(* Logix 5000 project; controller Y059_LHM vendor 1 type 14 code 156 rev 32.13; software revision 32.00 *)

TASK MainTask (periodic, rate 100 ms, priority 5, watchdog 500 ms) : MainProgram

MODULES
   Local : vendor 1 type 14 code 156 (Compact 0, rev 32.13)
      Module1 : 1769-IQ16 (Compact 1, rev 1.1, Input RPI 20 ms)
      Module2 : 1769-OB16 (Compact 2, rev 2.1, Output RPI 20 ms)
      SIC_101_Kinetix : vendor 1 type 37 code 50 (Ethernet 10.1.5.59, rev 7.11, MotionSync RPI 2 ms, MotionDiagnostics RPI 1 ms)
      SIC_201_Kinetix : vendor 1 type 37 code 50 (Ethernet 10.1.5.60, rev 7.1, MotionSync RPI 2 ms, MotionDiagnostics RPI 1 ms)
      Stratix5700 : vendor 1 type 12 code 242 (Ethernet 10.1.5.253, rev 10.1, Output RPI 1000 ms)
END_MODULES

TYPE Command :
STRUCT
   Command : DINT;   // 0=Run, 1=Fault Reset,
   Speed : REAL;   // Speed
END_STRUCT
END_TYPE

TYPE CommInfo :
STRUCT
   BoolTags : DINT;
   HeartBeat : DINT;
END_STRUCT
END_TYPE

TYPE FaultRecord :
STRUCT
   TimeLow : DINT;
   TimeHigh : DINT;
   Type : INT;
   Code : INT;
   Info : DINT[8];
END_STRUCT
END_TYPE

TYPE PumpController :
STRUCT
   RunCMD : BOOL;   // Run Command
   ResetCMD : BOOL;   // Reset Command
   isFaulted : BOOL;   // Fault Status, (0= Not Fault, 1= Faulted)
   isRunning : BOOL;   // Run Status, (0=Stopped, 1=Running)
   isServoOK : BOOL;   // Communications between the PLC and Servo (0=Not OK, 1=OK)
   isPressureHigh : BOOL;   // Outlet Pressure High Status (0=Not High, 1=High)
   isDecontactor : BOOL;   // Decontactor from STO circuit( 0=Contact OK, 1= Not Contact)
   FautCode : DINT;   // Fault Code
   SpeedSP : SetPoint;   // Speed Setpoint
   SpeedFeedback : SetPoint;   // Speed Feedback
   Ok2Run : BOOL;   // OK to Run Pump
   ResetTimer : TIMER;   // Heart Beat Error Reset Timer
END_STRUCT
END_TYPE

TYPE SetPoint :
STRUCT
   Min : REAL;
   SP : REAL;
   Max : REAL;
END_STRUCT
END_TYPE

TYPE Status :
STRUCT
   Status : DINT;   // 0=isDecontacted, 1=isFaulted, 2=isPressureHigh, 3=isRunning, 4=isServoOK
   FaultCode : DINT;
   SpeedFdbk : REAL;
END_STRUCT
END_TYPE

ADD_ON_INSTRUCTION SERVO_AOI   (* revision 1.0, vendor Lewa Process Technologies *)
// Servo AOI
// Help:
// Version 1.0
// 18 May, 2018
VAR_IN_OUT
   CONTROLLER : PumpController; {required}
   DRIVE_AXIS : AXIS_CIP_DRIVE; {required}
END_VAR
VAR_INPUT
   GearBox_Ratio : REAL; {access Read Only, required}   // GearBox Ratio (Read from Pump Name Plate)
   Axis_AccDec : REAL := 20.0; {required}
   Pump_RPM_Max : DINT; {access Read Only, required}
   Pump_RPM_Min : DINT; {access None, required}
END_VAR
VAR_OUTPUT
   Pump_RPM_Val : REAL; {access Read Only, visible}
   Motor_RPS : REAL; {visible}   // Speed RPS
END_VAR
VAR
   Local_Axis_MAFR : MOTION_INSTRUCTION;
   Local_Axis_MAJ : MOTION_INSTRUCTION;
   Local_Axis_MAS : MOTION_INSTRUCTION;
   Local_Axis_MCD : MOTION_INSTRUCTION;
   Local_Axis_MSF : MOTION_INSTRUCTION;
   Local_Axis_MSO : MOTION_INSTRUCTION;
   Motor_RPS_Prev : REAL;   // Previous Speed RPS
   Local_Axis_Start : BOOL;   // Servo Start/Stop Command
   Local_1000MaxRPM : DINT;   // 1000 Times Max RPM
   Local_RunDelay : TIMER := (PRE := 2000);
   Local_1000RPM : DINT; {access None}   // 1000 Times RPM
   Local_1000MinRPM : DINT; {access None}   // 1000 Times Min RPM
   ServoActualRPS : REAL; {access None}
   ServoActual : DINT; {access None}   // Motor RPS for Feedback
   Feedbk_1000RPM : DINT; {access None}   // 1000 Times RPM for Feedback
   Axis_Last_TrackingNotchFilter : REAL; {access None}
   Axis_NotchFilter_Seq : DINT; {access None}
   Axis_Timer : TIMER[4] := ([0].PRE := 50, [0].ACC := 60, [1].PRE := 50); {access None}
   Axis_CountUP : DINT; {access None}
   Axis_ONS0 : BOOL; {access None}
   Axis_AdaptiveTuning_Mode : DINT; {access None}
   Motor_RPS_ONS : BOOL; {access None}
END_VAR

ROUTINE Logic   (* ladder *)
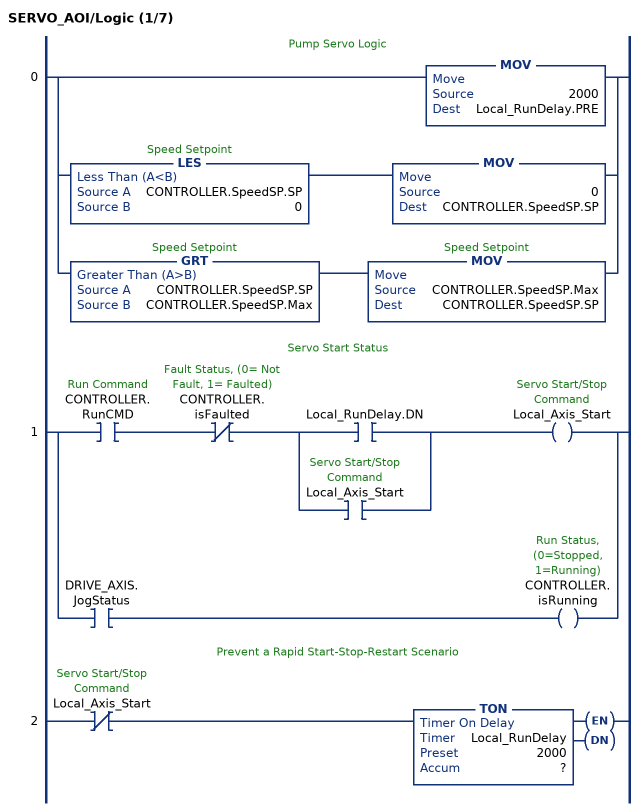
   // Pump Servo Logic
   0: [MOV(2000,Local_RunDelay.PRE) ,LES(CONTROLLER.SpeedSP.SP,0) MOV(0,CONTROLLER.SpeedSP.SP) ,GRT(CONTROLLER.SpeedSP.SP,CONTROLLER.SpeedSP.Max) MOV(CONTROLLER.SpeedSP.Max,CONTROLLER.SpeedSP.SP) ];
   // Servo Start Status
   1: [XIC(CONTROLLER.RunCMD) XIO(CONTROLLER.isFaulted) [XIC(Local_RunDelay.DN) ,XIC(Local_Axis_Start) ] OTE(Local_Axis_Start) ,XIC(DRIVE_AXIS.JogStatus) OTE(CONTROLLER.isRunning) ];
   // Prevent a Rapid Start-Stop-Restart Scenario
   2: XIO(Local_Axis_Start)TON(Local_RunDelay,?,?);
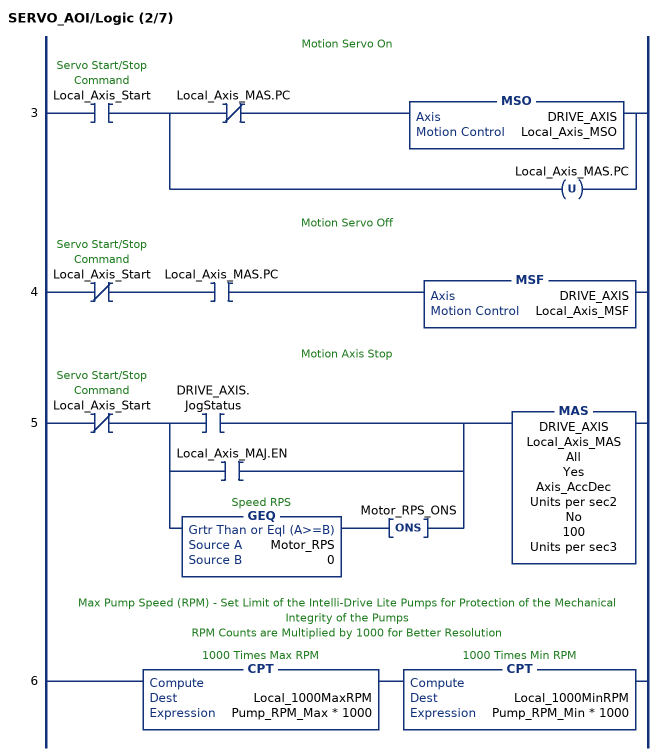
   // Motion Servo On
   3: XIC(Local_Axis_Start)[XIO(Local_Axis_MAS.PC) MSO(DRIVE_AXIS,Local_Axis_MSO) ,OTU(Local_Axis_MAS.PC) ];
   // Motion Servo Off
   4: XIO(Local_Axis_Start)XIC(Local_Axis_MAS.PC)MSF(DRIVE_AXIS,Local_Axis_MSF);
   // Motion Axis Stop
   5: XIO(Local_Axis_Start)[[XIC(DRIVE_AXIS.JogStatus) ,XIC(Local_Axis_MAJ.EN) ] ,GEQ(Motor_RPS,0) ONS(Motor_RPS_ONS) ]MAS(DRIVE_AXIS,Local_Axis_MAS,All,Yes,Axis_AccDec,Units per sec2,No,100,Units per sec3);
   // Max Pump Speed (RPM) - Set Limit of the Intelli-Drive Lite Pumps for Protection of the Mechanical Integrity of the Pumps
   // RPM Counts are Multiplied by 1000 for Better Resolution
   6: CPT(Local_1000MaxRPM,Pump_RPM_Max * 1000)CPT(Local_1000MinRPM,Pump_RPM_Min * 1000);
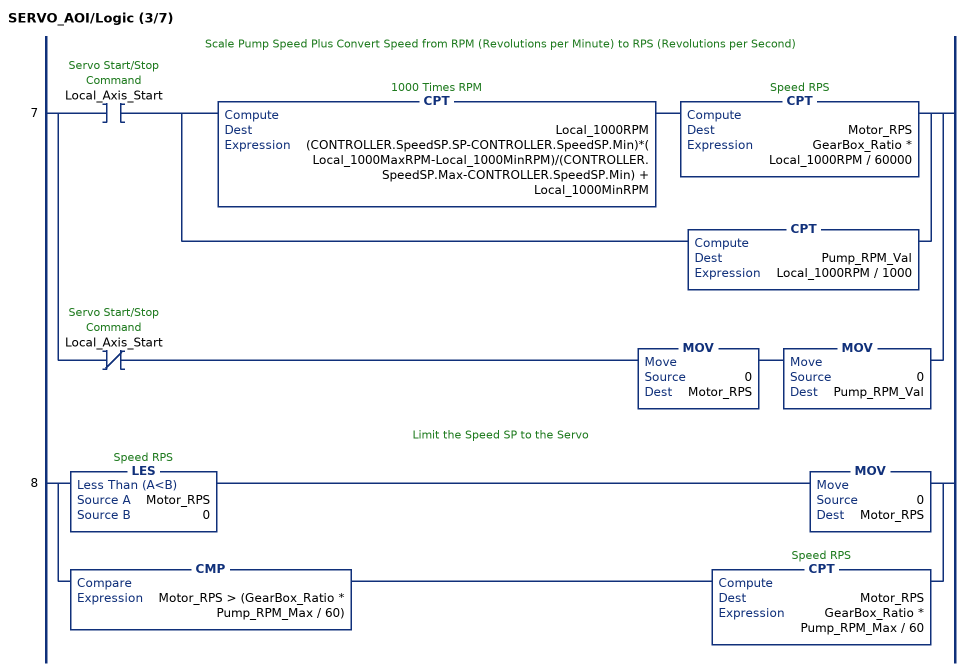
   // Scale Pump Speed Plus Convert Speed from RPM (Revolutions per Minute) to RPS (Revolutions per Second)
   7: [XIC(Local_Axis_Start) [CPT(Local_1000RPM,(CONTROLLER.SpeedSP.SP-CONTROLLER.SpeedSP.Min)*(Local_1000MaxRPM-Local_1000MinRPM)/(CONTROLLER.SpeedSP.Max-CONTROLLER.SpeedSP.Min) + Local_1000MinRPM) CPT(Motor_RPS,GearBox_Ratio * Local_1000RPM / 60000) ,CPT(Pump_RPM_Val,Local_1000RPM / 1000) ] ,XIO(Local_Axis_Start) MOV(0,Motor_RPS) MOV(0,Pump_RPM_Val) ];
   // Limit the Speed SP to the Servo
   8: [LES(Motor_RPS,0) MOV(0,Motor_RPS) ,CMP(Motor_RPS > (GearBox_Ratio * Pump_RPM_Max / 60)) CPT(Motor_RPS,GearBox_Ratio * Pump_RPM_Max / 60) ];
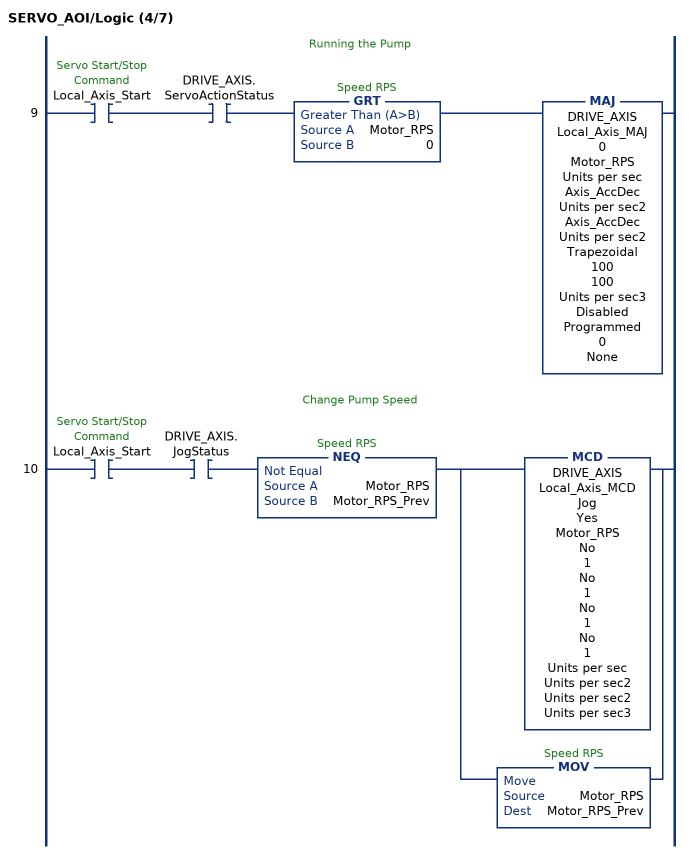
   // Running the Pump
   9: XIC(Local_Axis_Start)XIC(DRIVE_AXIS.ServoActionStatus)GRT(Motor_RPS,0)MAJ(DRIVE_AXIS,Local_Axis_MAJ,0,Motor_RPS,Units per sec,Axis_AccDec,Units per sec2,Axis_AccDec,Units per sec2,Trapezoidal,100,100,Units per sec3,Disabled,Programmed,0,None);
   // Change Pump Speed
   10: XIC(Local_Axis_Start)XIC(DRIVE_AXIS.JogStatus)NEQ(Motor_RPS,Motor_RPS_Prev)[MCD(DRIVE_AXIS,Local_Axis_MCD,Jog,Yes,Motor_RPS,No,1,No,1,No,1,No,1,Units per sec,Units per sec2,Units per sec2,Units per sec3) ,MOV(Motor_RPS,Motor_RPS_Prev) ];
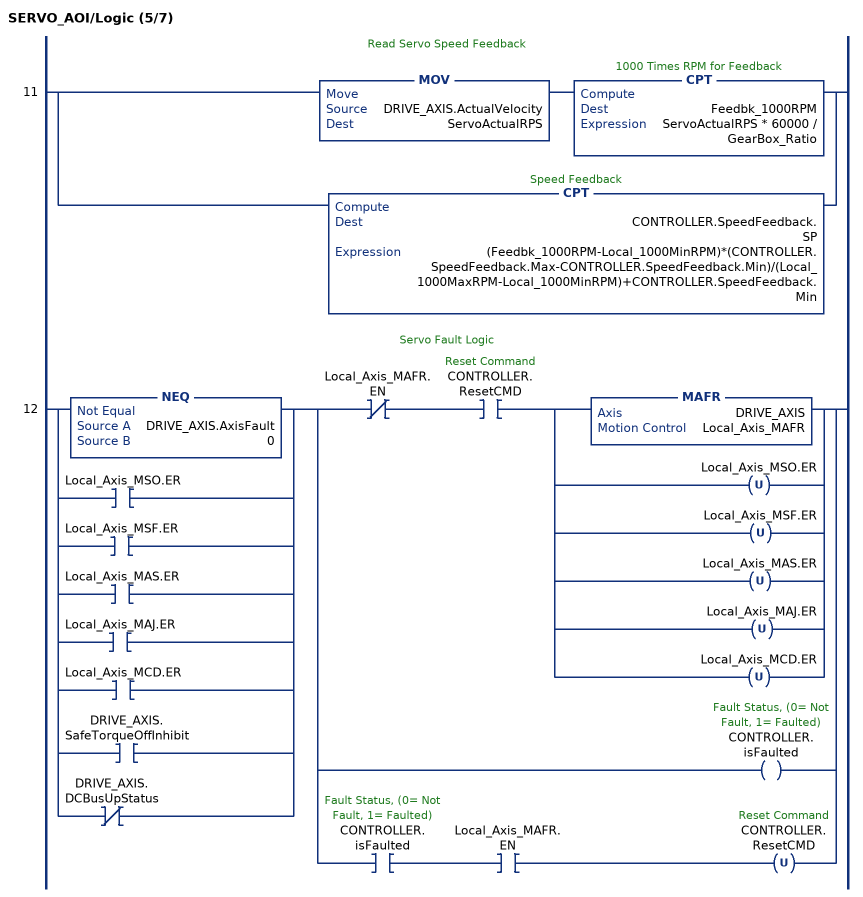
   // Read Servo Speed Feedback
   11: [MOV(DRIVE_AXIS.ActualVelocity,ServoActualRPS) CPT(Feedbk_1000RPM,ServoActualRPS * 60000 / GearBox_Ratio) ,CPT(CONTROLLER.SpeedFeedback.SP,(Feedbk_1000RPM-Local_1000MinRPM)*(CONTROLLER.SpeedFeedback.Max-CONTROLLER.SpeedFeedback.Min)/(Local_1000MaxRPM-Local_1000MinRPM)+CONTROLLER.SpeedFeedback.Min) ];
   // Servo Fault Logic
   12: [NEQ(DRIVE_AXIS.AxisFault,0) ,XIC(Local_Axis_MSO.ER) ,XIC(Local_Axis_MSF.ER) ,XIC(Local_Axis_MAS.ER) ,XIC(Local_Axis_MAJ.ER) ,XIC(Local_Axis_MCD.ER) ,XIC(DRIVE_AXIS.SafeTorqueOffInhibit) ,XIO(DRIVE_AXIS.DCBusUpStatus) ][XIO(Local_Axis_MAFR.EN) XIC(CONTROLLER.ResetCMD) [MAFR(DRIVE_AXIS,Local_Axis_MAFR) ,OTU(Local_Axis_MSO.ER) ,OTU(Local_Axis_MSF.ER) ,OTU(Local_Axis_MAS.ER) ,OTU(Local_Axis_MAJ.ER) ,OTU(Local_Axis_MCD.ER) ] ,OTE(CONTROLLER.isFaulted) ,XIC(CONTROLLER.isFaulted) XIC(Local_Axis_MAFR.EN) OTU(CONTROLLER.ResetCMD) ];
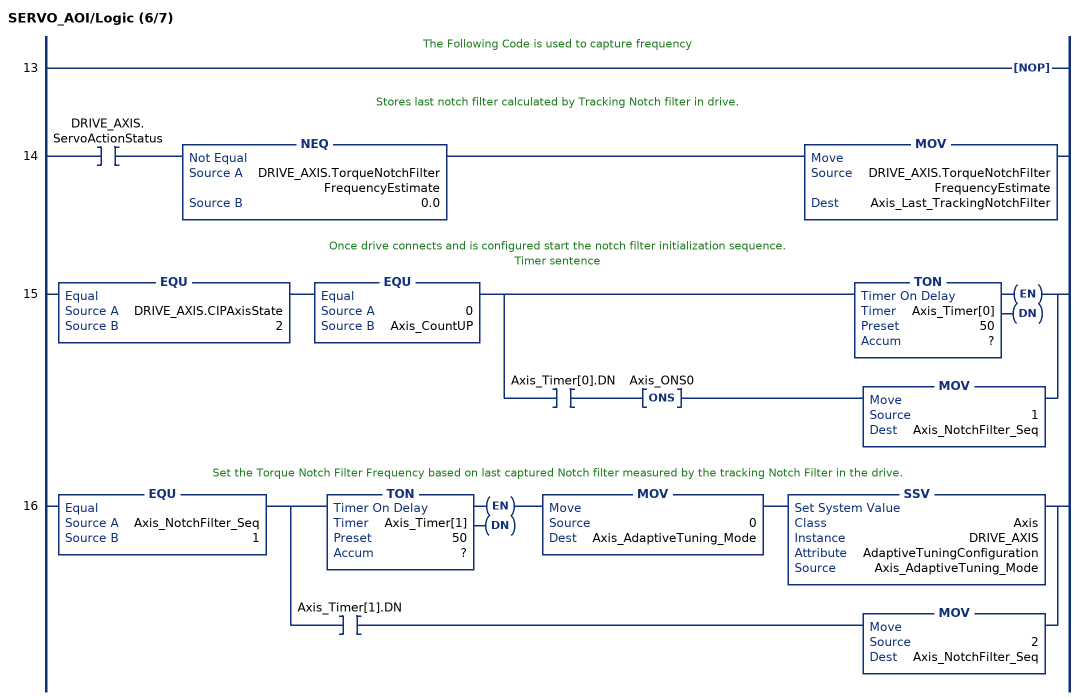
   // The Following Code is used to capture frequency
   13: NOP();
   // Stores last notch filter calculated by Tracking Notch filter in drive.
   14: XIC(DRIVE_AXIS.ServoActionStatus)NEQ(DRIVE_AXIS.TorqueNotchFilterFrequencyEstimate,0.0)MOV(DRIVE_AXIS.TorqueNotchFilterFrequencyEstimate,Axis_Last_TrackingNotchFilter);
   // Once drive connects and is configured start the notch filter initialization sequence.
   // Timer sentence
   15: EQU(DRIVE_AXIS.CIPAxisState,2)EQU(0,Axis_CountUP)[TON(Axis_Timer[0],?,?) ,XIC(Axis_Timer[0].DN) ONS(Axis_ONS0) MOV(1,Axis_NotchFilter_Seq) ];
   // Set the Torque Notch Filter Frequency based on last captured Notch filter measured by the tracking Notch Filter in the drive.
   16: EQU(Axis_NotchFilter_Seq,1)[TON(Axis_Timer[1],?,?) MOV(0,Axis_AdaptiveTuning_Mode) SSV(Axis,DRIVE_AXIS,AdaptiveTuningConfiguration,Axis_AdaptiveTuning_Mode) ,XIC(Axis_Timer[1].DN) MOV(2,Axis_NotchFilter_Seq) ];
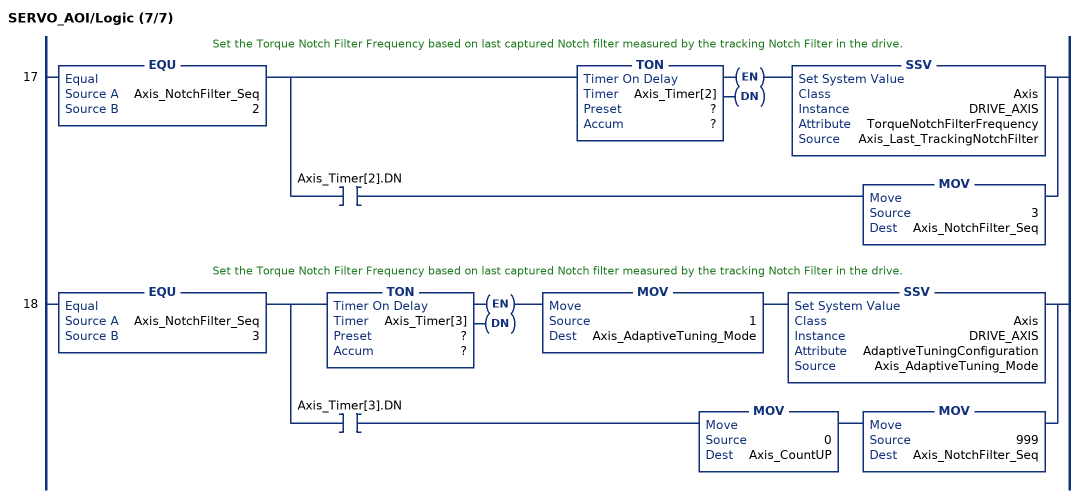
   // Set the Torque Notch Filter Frequency based on last captured Notch filter measured by the tracking Notch Filter in the drive.
   17: EQU(Axis_NotchFilter_Seq,2)[TON(Axis_Timer[2],?,?) SSV(Axis,DRIVE_AXIS,TorqueNotchFilterFrequency,Axis_Last_TrackingNotchFilter) ,XIC(Axis_Timer[2].DN) MOV(3,Axis_NotchFilter_Seq) ];
   // Set the Torque Notch Filter Frequency based on last captured Notch filter measured by the tracking Notch Filter in the drive.
   18: EQU(Axis_NotchFilter_Seq,3)[TON(Axis_Timer[3],?,?) MOV(1,Axis_AdaptiveTuning_Mode) SSV(Axis,DRIVE_AXIS,AdaptiveTuningConfiguration,Axis_AdaptiveTuning_Mode) ,XIC(Axis_Timer[3].DN) MOV(0,Axis_CountUP) MOV(999,Axis_NotchFilter_Seq) ];
END_ROUTINE
END_ADD_ON_INSTRUCTION

ADD_ON_INSTRUCTION ServoFaultCode   (* revision 1.0, vendor YMC Process Technologies *)
VAR_IN_OUT
   Axis_1 : AXIS_CIP_DRIVE; {required}
END_VAR
VAR_INPUT
   DriveConnStatus : DINT := 16#0000_4000; {required}
END_VAR
VAR_OUTPUT
   FaultCode : DINT; {access Read Only, required}
   FaultType : DINT; {access Read Only, required}
   LocalFaultDetected : BOOL; {access None, required}
END_VAR
VAR
   A1_CIPAxisFaultsLSW : DINT;
   A1_CIPAxisFaultsMSW : DINT := 45;
   A1_CIPAxisFaultsRA_LSW : DINT;
   A1_CIPAxisFaultsRA_MSW : DINT;
   ErrorCode : DINT[20] := ([1] := 8192);
   IntegratedSTOSxx : DINT; {access None}
   A1_AxisSafetyFaults : DINT; {access None}
   Drive_CommConnectionOK : BOOL; {access None}
   TempCipAxisFaultsRA : DINT[2]; {access None}
   ClearFault : DINT; {access None}
END_VAR

ROUTINE Logic   (* ladder *)
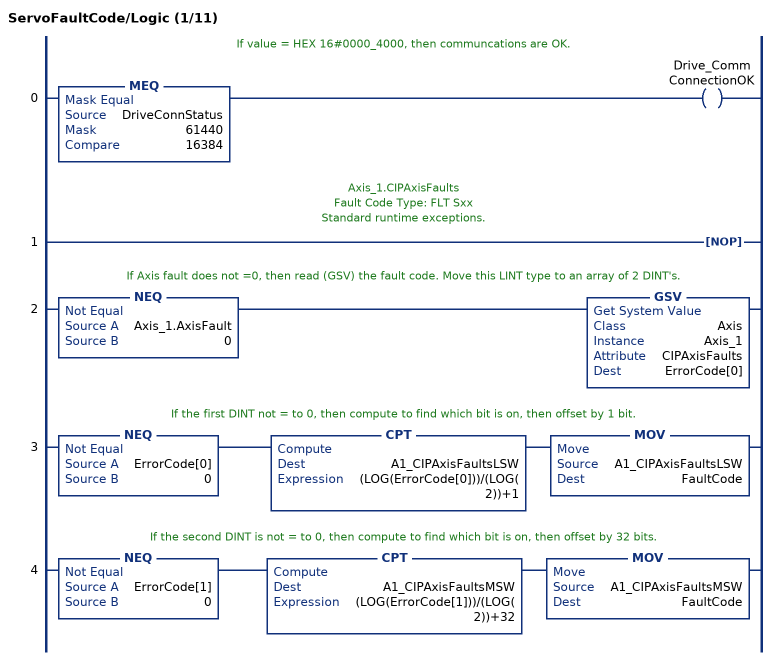
   // If value = HEX 16#0000_4000, then communcations are OK.
   0: MEQ(DriveConnStatus,61440,16384)OTE(Drive_CommConnectionOK);
   // Axis_1.CIPAxisFaults
   // Fault Code Type: FLT Sxx
   // Standard runtime exceptions.
   1: NOP();
   // If Axis fault does not =0, then read (GSV) the fault code. Move this LINT type to an array of 2 DINT's.
   2: NEQ(Axis_1.AxisFault,0)GSV(Axis,Axis_1,CIPAxisFaults,ErrorCode[0]);
   // If the first DINT not = to 0, then compute to find which bit is on, then offset by 1 bit.
   3: NEQ(ErrorCode[0],0)CPT(A1_CIPAxisFaultsLSW,(LOG(ErrorCode[0]))/(LOG(2))+1)MOV(A1_CIPAxisFaultsLSW,FaultCode);
   // If the second DINT is not = to 0, then compute to find which bit is on, then offset by 32 bits.
   4: NEQ(ErrorCode[1],0)CPT(A1_CIPAxisFaultsMSW,(LOG(ErrorCode[1]))/(LOG(2))+32)MOV(A1_CIPAxisFaultsMSW,FaultCode);
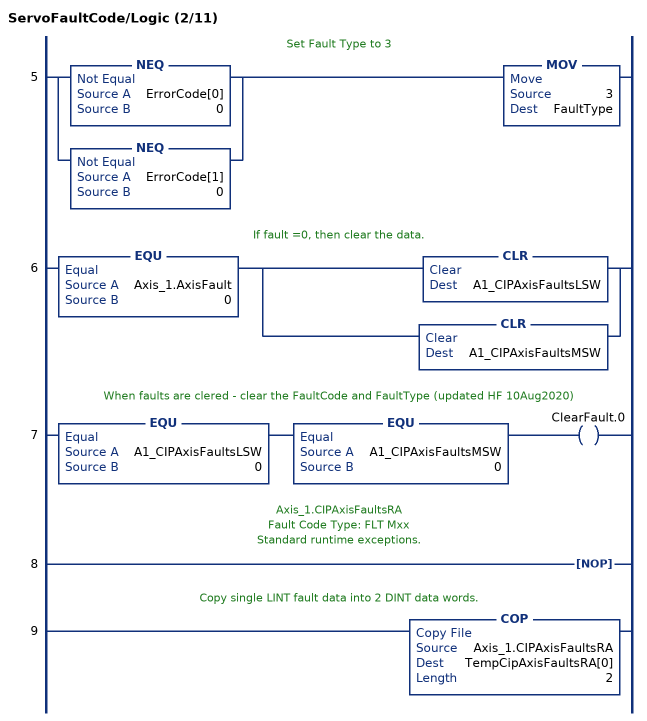
   // Set Fault Type to 3
   5: [NEQ(ErrorCode[0],0) ,NEQ(ErrorCode[1],0) ]MOV(3,FaultType);
   // If fault =0, then clear the data.
   6: EQU(Axis_1.AxisFault,0)[CLR(A1_CIPAxisFaultsLSW) ,CLR(A1_CIPAxisFaultsMSW) ];
   // When faults are clered - clear the FaultCode and FaultType (updated HF 10Aug2020)
   7: EQU(A1_CIPAxisFaultsLSW,0)EQU(A1_CIPAxisFaultsMSW,0)OTE(ClearFault.0);
   // Axis_1.CIPAxisFaultsRA
   // Fault Code Type: FLT Mxx
   // Standard runtime exceptions.
   8: NOP();
   // Copy single LINT fault data into 2 DINT data words.
   9: COP(Axis_1.CIPAxisFaultsRA,TempCipAxisFaultsRA[0],2);
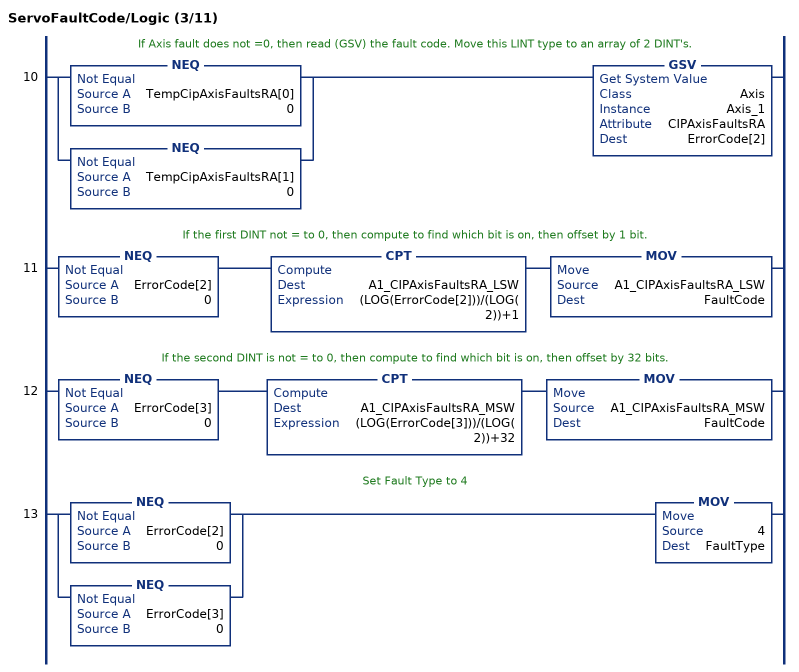
   // If Axis fault does not =0, then read (GSV) the fault code. Move this LINT type to an array of 2 DINT's.
   10: [NEQ(TempCipAxisFaultsRA[0],0) ,NEQ(TempCipAxisFaultsRA[1],0) ]GSV(Axis,Axis_1,CIPAxisFaultsRA,ErrorCode[2]);
   // If the first DINT not = to 0, then compute to find which bit is on, then offset by 1 bit.
   11: NEQ(ErrorCode[2],0)CPT(A1_CIPAxisFaultsRA_LSW,(LOG(ErrorCode[2]))/(LOG(2))+1)MOV(A1_CIPAxisFaultsRA_LSW,FaultCode);
   // If the second DINT is not = to 0, then compute to find which bit is on, then offset by 32 bits.
   12: NEQ(ErrorCode[3],0)CPT(A1_CIPAxisFaultsRA_MSW,(LOG(ErrorCode[3]))/(LOG(2))+32)MOV(A1_CIPAxisFaultsRA_MSW,FaultCode);
   // Set Fault Type to 4
   13: [NEQ(ErrorCode[2],0) ,NEQ(ErrorCode[3],0) ]MOV(4,FaultType);
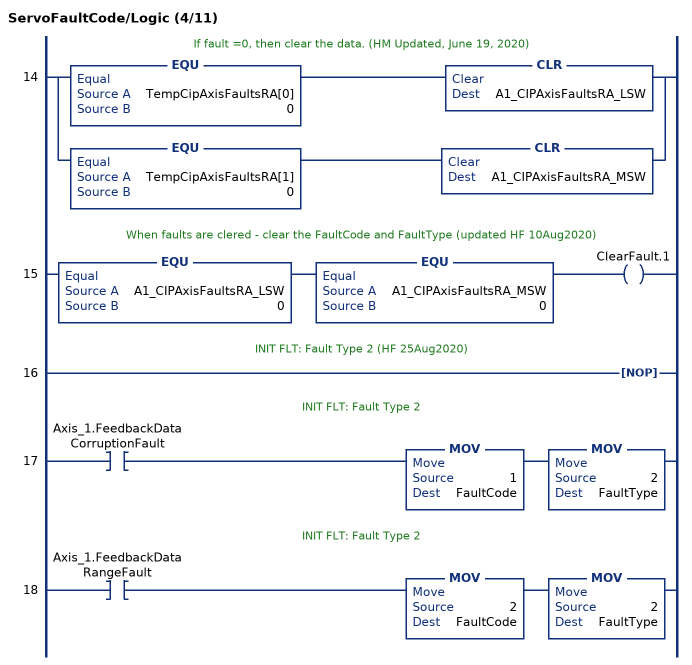
   // If fault =0, then clear the data. (HM Updated, June 19, 2020)
   14: [EQU(TempCipAxisFaultsRA[0],0) CLR(A1_CIPAxisFaultsRA_LSW) ,EQU(TempCipAxisFaultsRA[1],0) CLR(A1_CIPAxisFaultsRA_MSW) ];
   // When faults are clered - clear the FaultCode and FaultType (updated HF 10Aug2020)
   15: EQU(A1_CIPAxisFaultsRA_LSW,0)EQU(A1_CIPAxisFaultsRA_MSW,0)OTE(ClearFault.1);
   // INIT FLT: Fault Type 2 (HF 25Aug2020)
   16: NOP();
   // INIT FLT: Fault Type 2
   17: XIC(Axis_1.FeedbackDataCorruptionFault)MOV(1,FaultCode)MOV(2,FaultType);
   // INIT FLT: Fault Type 2
   18: XIC(Axis_1.FeedbackDataRangeFault)MOV(2,FaultCode)MOV(2,FaultType);
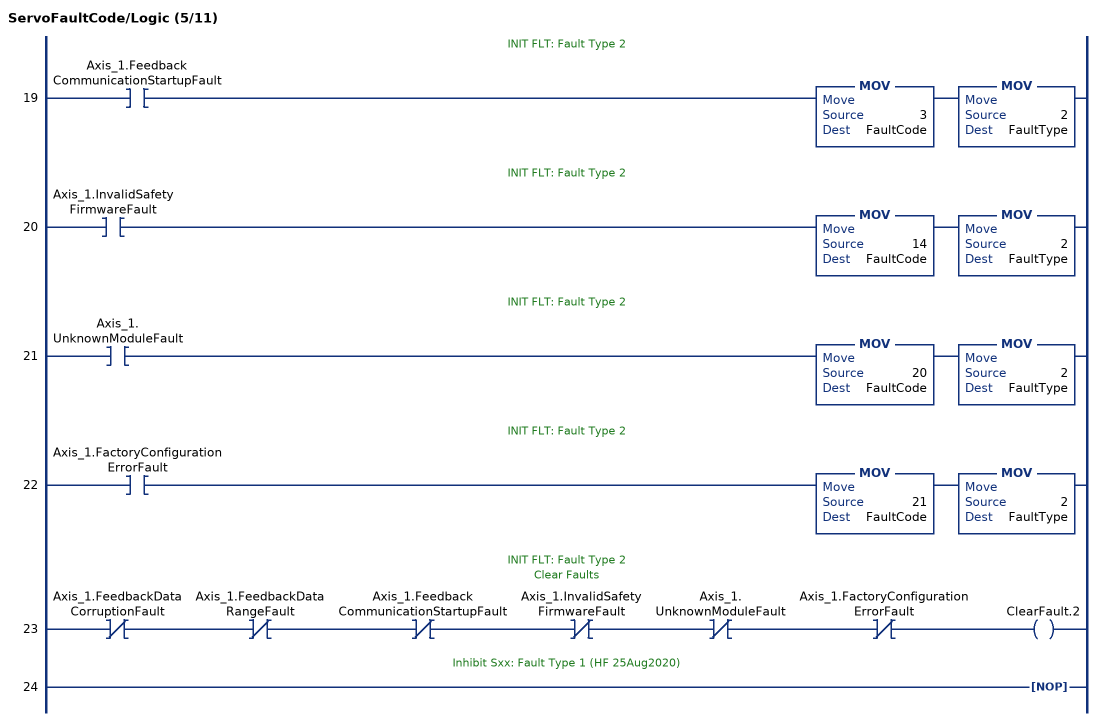
   // INIT FLT: Fault Type 2
   19: XIC(Axis_1.FeedbackCommunicationStartupFault)MOV(3,FaultCode)MOV(2,FaultType);
   // INIT FLT: Fault Type 2
   20: XIC(Axis_1.InvalidSafetyFirmwareFault)MOV(14,FaultCode)MOV(2,FaultType);
   // INIT FLT: Fault Type 2
   21: XIC(Axis_1.UnknownModuleFault)MOV(20,FaultCode)MOV(2,FaultType);
   // INIT FLT: Fault Type 2
   22: XIC(Axis_1.FactoryConfigurationErrorFault)MOV(21,FaultCode)MOV(2,FaultType);
   // INIT FLT: Fault Type 2
   // Clear Faults
   23: XIO(Axis_1.FeedbackDataCorruptionFault)XIO(Axis_1.FeedbackDataRangeFault)XIO(Axis_1.FeedbackCommunicationStartupFault)XIO(Axis_1.InvalidSafetyFirmwareFault)XIO(Axis_1.UnknownModuleFault)XIO(Axis_1.FactoryConfigurationErrorFault)OTE(ClearFault.2);
   // Inhibit Sxx: Fault Type 1 (HF 25Aug2020)
   24: NOP();
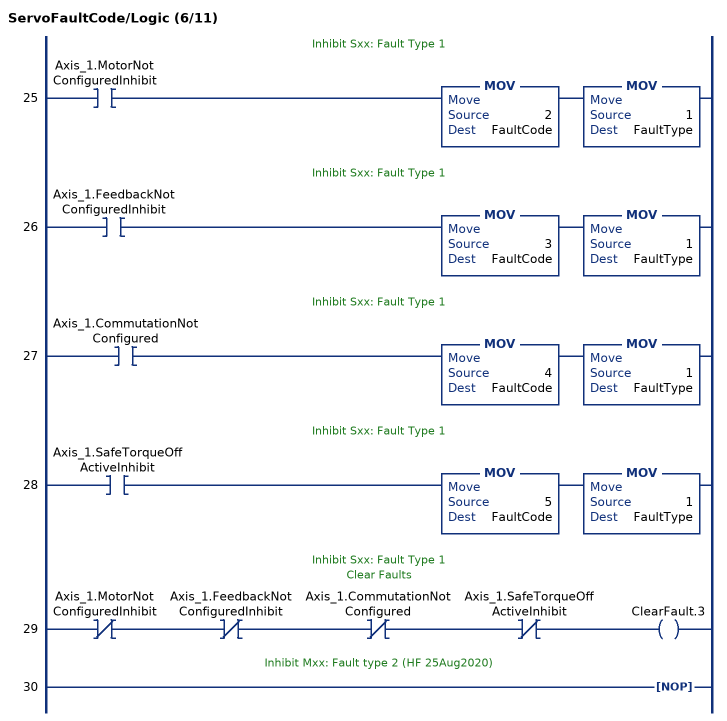
   // Inhibit Sxx: Fault Type 1
   25: XIC(Axis_1.MotorNotConfiguredInhibit)MOV(2,FaultCode)MOV(1,FaultType);
   // Inhibit Sxx: Fault Type 1
   26: XIC(Axis_1.FeedbackNotConfiguredInhibit)MOV(3,FaultCode)MOV(1,FaultType);
   // Inhibit Sxx: Fault Type 1
   27: XIC(Axis_1.CommutationNotConfigured)MOV(4,FaultCode)MOV(1,FaultType);
   // Inhibit Sxx: Fault Type 1
   28: XIC(Axis_1.SafeTorqueOffActiveInhibit)MOV(5,FaultCode)MOV(1,FaultType);
   // Inhibit Sxx: Fault Type 1
   // Clear Faults
   29: XIO(Axis_1.MotorNotConfiguredInhibit)XIO(Axis_1.FeedbackNotConfiguredInhibit)XIO(Axis_1.CommutationNotConfigured)XIO(Axis_1.SafeTorqueOffActiveInhibit)OTE(ClearFault.3);
   // Inhibit Mxx: Fault type 2 (HF 25Aug2020)
   30: NOP();
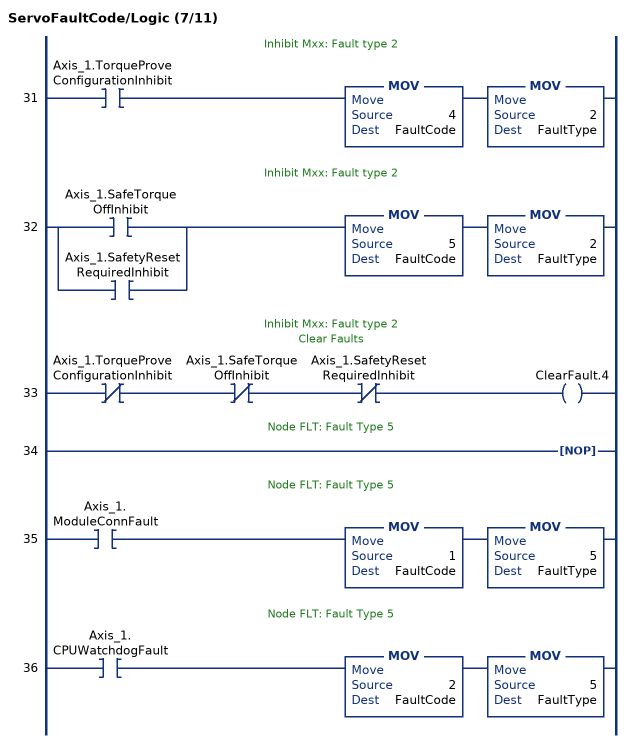
   // Inhibit Mxx: Fault type 2
   31: XIC(Axis_1.TorqueProveConfigurationInhibit)MOV(4,FaultCode)MOV(2,FaultType);
   // Inhibit Mxx: Fault type 2
   32: [XIC(Axis_1.SafeTorqueOffInhibit) ,XIC(Axis_1.SafetyResetRequiredInhibit) ]MOV(5,FaultCode)MOV(2,FaultType);
   // Inhibit Mxx: Fault type 2
   // Clear Faults
   33: XIO(Axis_1.TorqueProveConfigurationInhibit)XIO(Axis_1.SafeTorqueOffInhibit)XIO(Axis_1.SafetyResetRequiredInhibit)OTE(ClearFault.4);
   // Node FLT: Fault Type 5
   34: NOP();
   // Node FLT: Fault Type 5
   35: XIC(Axis_1.ModuleConnFault)MOV(1,FaultCode)MOV(5,FaultType);
   // Node FLT: Fault Type 5
   36: XIC(Axis_1.CPUWatchdogFault)MOV(2,FaultCode)MOV(5,FaultType);
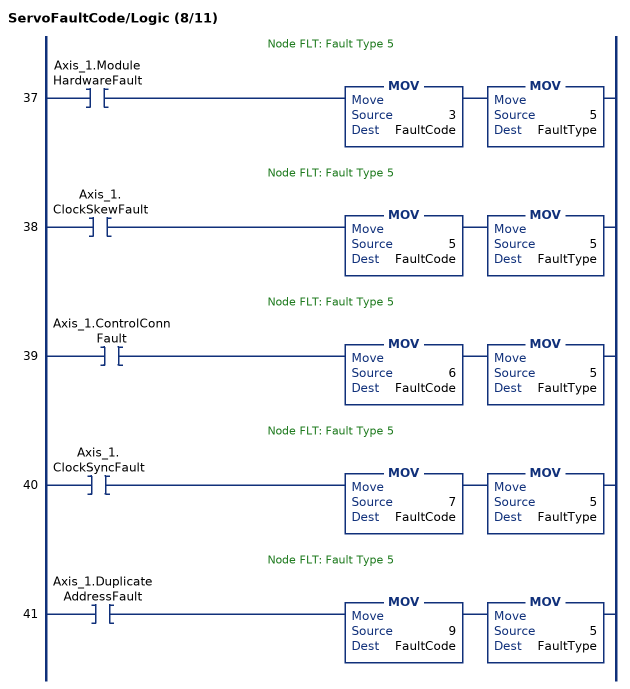
   // Node FLT: Fault Type 5
   37: XIC(Axis_1.ModuleHardwareFault)MOV(3,FaultCode)MOV(5,FaultType);
   // Node FLT: Fault Type 5
   38: XIC(Axis_1.ClockSkewFault)MOV(5,FaultCode)MOV(5,FaultType);
   // Node FLT: Fault Type 5
   39: XIC(Axis_1.ControlConnFault)MOV(6,FaultCode)MOV(5,FaultType);
   // Node FLT: Fault Type 5
   40: XIC(Axis_1.ClockSyncFault)MOV(7,FaultCode)MOV(5,FaultType);
   // Node FLT: Fault Type 5
   41: XIC(Axis_1.DuplicateAddressFault)MOV(9,FaultCode)MOV(5,FaultType);
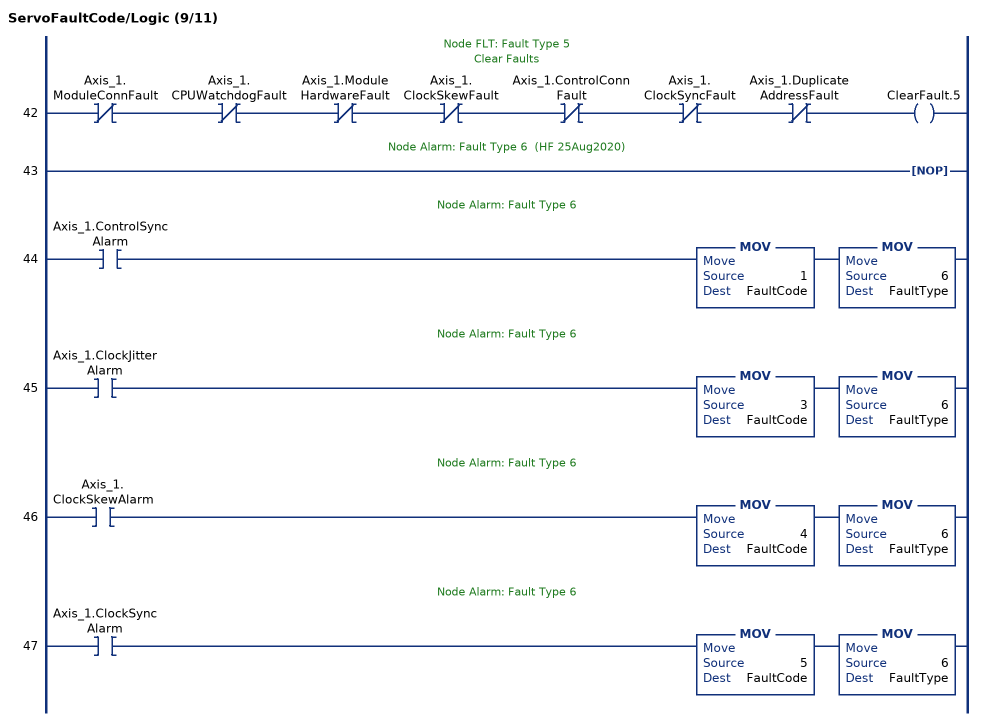
   // Node FLT: Fault Type 5
   // Clear Faults
   42: XIO(Axis_1.ModuleConnFault)XIO(Axis_1.CPUWatchdogFault)XIO(Axis_1.ModuleHardwareFault)XIO(Axis_1.ClockSkewFault)XIO(Axis_1.ControlConnFault)XIO(Axis_1.ClockSyncFault)XIO(Axis_1.DuplicateAddressFault)OTE(ClearFault.5);
   // Node Alarm: Fault Type 6  (HF 25Aug2020)
   43: NOP();
   // Node Alarm: Fault Type 6
   44: XIC(Axis_1.ControlSyncAlarm)MOV(1,FaultCode)MOV(6,FaultType);
   // Node Alarm: Fault Type 6
   45: XIC(Axis_1.ClockJitterAlarm)MOV(3,FaultCode)MOV(6,FaultType);
   // Node Alarm: Fault Type 6
   46: XIC(Axis_1.ClockSkewAlarm)MOV(4,FaultCode)MOV(6,FaultType);
   // Node Alarm: Fault Type 6
   47: XIC(Axis_1.ClockSyncAlarm)MOV(5,FaultCode)MOV(6,FaultType);
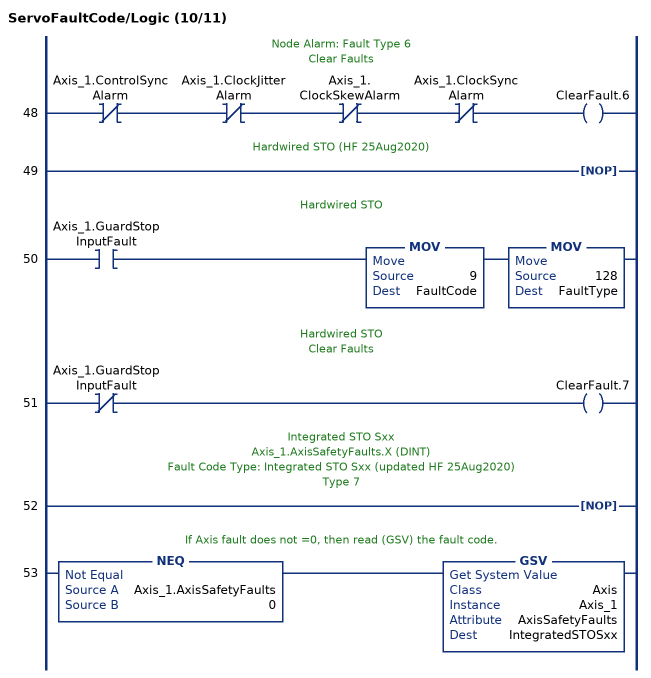
   // Node Alarm: Fault Type 6
   // Clear Faults
   48: XIO(Axis_1.ControlSyncAlarm)XIO(Axis_1.ClockJitterAlarm)XIO(Axis_1.ClockSkewAlarm)XIO(Axis_1.ClockSyncAlarm)OTE(ClearFault.6);
   // Hardwired STO (HF 25Aug2020)
   49: NOP();
   // Hardwired STO
   50: XIC(Axis_1.GuardStopInputFault)MOV(9,FaultCode)MOV(128,FaultType);
   // Hardwired STO
   // Clear Faults
   51: XIO(Axis_1.GuardStopInputFault)OTE(ClearFault.7);
   // Integrated STO Sxx
   // Axis_1.AxisSafetyFaults.X (DINT)
   // Fault Code Type: Integrated STO Sxx (updated HF 25Aug2020)
   // Type 7
   52: NOP();
   // If Axis fault does not =0, then read (GSV) the fault code.
   53: NEQ(Axis_1.AxisSafetyFaults,0)GSV(Axis,Axis_1,AxisSafetyFaults,IntegratedSTOSxx);
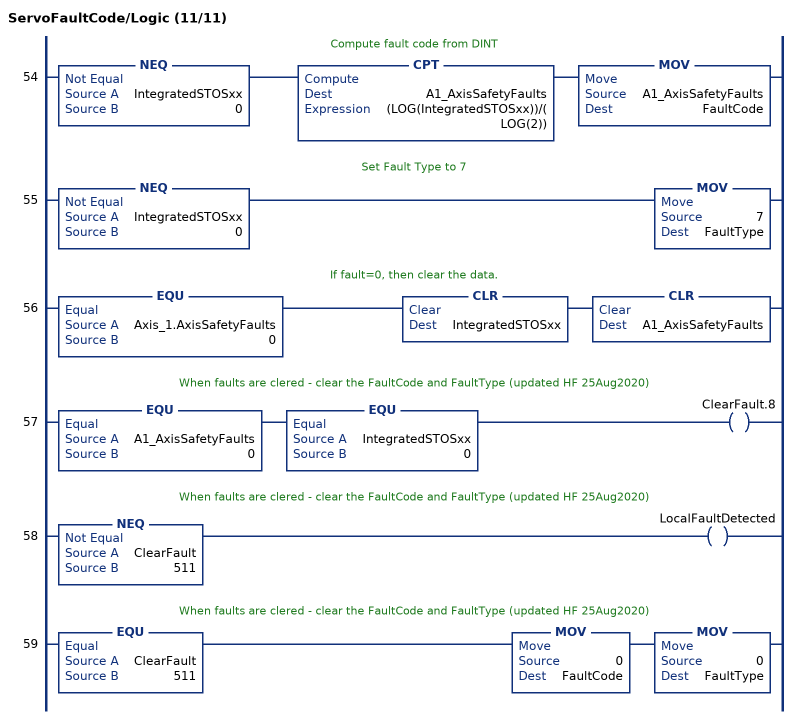
   // Compute fault code from DINT
   54: NEQ(IntegratedSTOSxx,0)CPT(A1_AxisSafetyFaults,(LOG(IntegratedSTOSxx))/(LOG(2)))MOV(A1_AxisSafetyFaults,FaultCode);
   // Set Fault Type to 7
   55: NEQ(IntegratedSTOSxx,0)MOV(7,FaultType);
   // If fault=0, then clear the data.
   56: EQU(Axis_1.AxisSafetyFaults,0)CLR(IntegratedSTOSxx)CLR(A1_AxisSafetyFaults);
   // When faults are clered - clear the FaultCode and FaultType (updated HF 25Aug2020)
   57: EQU(A1_AxisSafetyFaults,0)EQU(IntegratedSTOSxx,0)OTE(ClearFault.8);
   // When faults are clered - clear the FaultCode and FaultType (updated HF 25Aug2020)
   58: NEQ(ClearFault,511)OTE(LocalFaultDetected);
   // When faults are clered - clear the FaultCode and FaultType (updated HF 25Aug2020)
   59: EQU(ClearFault,511)MOV(0,FaultCode)MOV(0,FaultType);
END_ROUTINE
END_ADD_ON_INSTRUCTION
